INTERFACE I_Axis EXTENDS I_Cyclic

PROPERTY PUBLIC Acceleration : mc_lreal
GET
END_GET
SET
END_SET
END_PROPERTY

PROPERTY AxisRef : reference to Axis_Ref
GET
END_GET
END_PROPERTY

PROPERTY BufferMode : MC_BufferMode
GET
END_GET
SET
END_SET
END_PROPERTY

PROPERTY PUBLIC Deceleration : mc_lreal
GET
END_GET
SET
END_SET
END_PROPERTY

METHOD PUBLIC DisableAxis : HRESULT
VAR_INPUT
END_VAR
END_METHOD

METHOD PUBLIC EnableAxis : HRESULT
VAR_INPUT
	InhibitPositive : BOOL;
	InhibitNegative : BOOL;
END_VAR
END_METHOD

PROPERTY ErrorID : DWORD
GET
END_GET
END_PROPERTY

METHOD PUBLIC HaltAxis : HRESULT
VAR
END_VAR
END_METHOD

PROPERTY PUBLIC Jerk : mc_lreal
GET
END_GET
SET
END_SET
END_PROPERTY

PROPERTY Operating : BOOL
GET
END_GET
END_PROPERTY

METHOD PUBLIC Reset : HRESULT
VAR
END_VAR
END_METHOD

END_INTERFACE

(* stored: Version 1.1.0.1
   Itf I_Axis: Id {0ef07e09-d612-4b35-8507-c5527a9d7e82}
   Property Acceleration: Id {72d27c44-987d-44ce-a99c-48cb32673553}
   Get Get: Id {056425fd-3278-4643-be11-9a6970fe13ef}
   Set Set: Id {9650a87b-bd43-4b24-b18c-102d81cc67c2}
   Property AxisRef: Id {e4c93f09-4784-43f3-989e-ffe0dbb5d4d1}
   Get Get: Id {43115712-1524-4aec-841c-f993969891f9}
   Property BufferMode: Id {84cb34ca-cf7c-44e5-808a-d05b61db3bfb}
   Get Get: Id {9281d6e3-005d-411b-9675-57d36646c8ee}
   Set Set: Id {9446d1c2-9a48-41b1-ba0a-d81d5dd2668a}
   Property Deceleration: Id {5ef3957c-6644-426d-8ede-03dbef11af09}
   Get Get: Id {bffc68c4-d0c8-4caa-bb08-1acb04f5a311}
   Set Set: Id {615e48f2-1833-4891-bf53-66cbe72eae8a}
   Method DisableAxis: Id {9aa78aa4-6937-4925-a0b3-e6b55191b9b8}
   Method EnableAxis: Id {1d051842-9ad9-43b4-9c63-942a1b02943c}
   Property ErrorID: Id {52b85bd9-c966-4845-b532-20088e4690ea}
   Get Get: Id {4d938dee-d107-459d-86cd-329dbada6b63}
   Method HaltAxis: Id {f00a986d-e8a1-4ddc-8d6f-7dfd0ff96b72}
   Property Jerk: Id {dd32e94c-e653-4f44-ba1a-16a122c64a8f}
   Get Get: Id {ed85520a-8680-4906-88bb-bb44509a959d}
   Set Set: Id {4339837f-910b-4c9c-913e-e3f9f3195613}
   Property Operating: Id {1989e548-414f-4241-9325-26b5e3866acf}
   Get Get: Id {ab90dda6-37af-4cff-9da4-9572d37a36e8}
   Method Reset: Id {70c30306-2843-45ea-9390-dee5671086b2} *)
